(* CoDeSys 2.3.9.62 project: AperturaConClave.pro *)
(* Libraries: Standard.lib 2.6.14 11:37:46 *)

(* Global variable list: Global_Variables *)
VAR_GLOBAL

   (* Entradas *)
  (* Botonera de entrada *)
   Ent1:BOOL;
   Ent2:BOOL;
   Ent3:BOOL;
   Ent4:BOOL;
   Cierre:BOOL;


   (* Salidas *)
   CajaAbierta: BOOL;

   (*Claves *)
   Clave1:INT:=1;
  Clave2:INT:=2;
  Clave3:INT:=2;


END_VAR

(* POU PLC_PRG, ST *)
PROGRAM PLC_PRG
VAR
(*Necesitamos un tof*)
	Tempo:TOF;
	E0,E1,E2,E3,E4,E5:BOOL;
	ValorInt:INT;
(**)
END_VAR
ValorInt := Decodificador(Ent1,Ent2, Ent3,Ent4);
Tempo.
IF NOT (E0  OR E1 OR E2 OR E3 ) THEN
E0 := TRUE;
ELSIF ValorInt = 0 THEN(* si no se ha pulsado ningún botón*)
E5:= E5;(* por poner *)
ELSIF (E0 AND Clave1= ValorInt) THEN  (*si estamos en E0 y la clave introducida es correcta *)
E0:= FALSE;
E1:=TRUE;
ELSIF E0 AND NOT (Clave1= ValorInt) THEN	(*si estamos en E0 y la clave introducida esin correcta(redundante) *)
E0:= FALSE;
E1:= TRUE;
ELSIF E1 AND Clave2= ValorInt THEN  (*si estamos en E1 y la clave introducida es correcta *)
E1:= FALSE;
E2:=TRUE;
ELSIF E1 AND NOT (Clave2= ValorInt) THEN	(*si estamos en E1 y la clave introducida esin correcta *)
E1:= FALSE;
E0:= TRUE;
ELSIF E2 AND Clave3= ValorInt THEN  (*si estamos en E1 y la clave introducida es correcta *)
E2:= FALSE;
E3:=TRUE;
ELSIF E2 AND NOT (Clave3= ValorInt) THEN	(*si estamos en E1 y la clave introducida esin correcta) *)
E2:= FALSE;
E0:= TRUE;
ELSIF E3 AND NOT Cierre THEN
CajaAbierta := TRUE;
E3 := TRUE;
E0:= FALSE;
ELSIF E3 AND  Cierre THEN
CajaAbierta := FALSE;
E3 := FALSE;
E0:= TRUE;
END_IF;
END_PROGRAM

(* POU Decodificador, ST *)
FUNCTION Decodificador : INT
VAR_INPUT
	E1:BOOL;
	E2:BOOL;
	E3:BOOL;
	E4:BOOL;
END_VAR
VAR
END_VAR
IF E1 = TRUE THEN
Decodificador := 1;
ELSIF E2 = TRUE THEN
Decodificador := 2;
ELSIF E3=TRUE THEN
Decodificador := 3;
ELSIF E4=TRUE THEN
Decodificador := 4;
ELSE
Decodificador := 0;
END_IF;
END_FUNCTION

(* Visualisation Visu
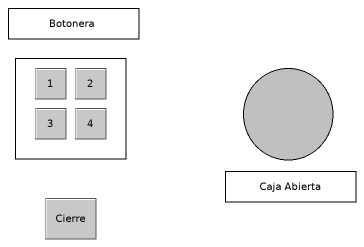
button at (50,130)-(81,161): text "1"; taps Ent1
button at (90,130)-(121,161): text "2"; taps Ent2
button at (50,170)-(81,201): text "3"; taps Ent3
button at (90,170)-(121,201): text "4"; taps Ent4
button at (60,260)-(111,301): text "Cierre"; taps Cierre
rectangle at (23,70)-(154,101): text "Botonera"
ellipse at (258,130)-(348,222): alarm colour if CajaAbierta
rectangle at (240,233)-(371,264): text "Caja Abierta"
1 more shapes without text or variables
*)
